DATA_BLOCK "DB3_CHECKSUM"
{ S7_Optimized_Access := 'TRUE' }
AUTHOR : AketzaBarragues
FAMILY : ZeusControl
VERSION : 1.0
NON_RETAIN
"FB3_ZC_CHECKSUM"

BEGIN

END_DATA_BLOCK

